Staubli VAL3: trajBuffer.pgx

public program trajBuffer(num x_nElems, num x_nPtsPopped)
begin

  // update trajectory buffer size

  userPageSet("uxMonitor", "lblTrajectoryBuffer", "innerHTML", x_nElems)
  userPageSet("uxMonitor", "lblTrajectoryBufferPopped", "innerHTML", x_nPtsPopped)

end
